TYPE typeMotionRowArry :
STRUCT
	data: ARRAY[1..99] OF typeMotionRecordRow;
END_STRUCT
END_TYPE

(* stored: Version 1.1.0.1, ProductVersion 3.1.4024.12
   DUT typeMotionRowArry: Id {c676dbe5-b639-4097-9ee3-56ef4cf4dac2} *)
